TYPE typeAutoRowMotion :
STRUCT
	Request:BOOL; //request the motion
	Depth:BOOL; //depth of the motion
	stepNumber:UINT; //step number, relates to left and right number on each row (option)
END_STRUCT
END_TYPE

(* stored: Version 1.1.0.1, ProductVersion 3.1.4024.11
   DUT typeAutoRowMotion: Id {187de1ff-1d9c-0c8b-24ec-085a1df2ebd5} *)
